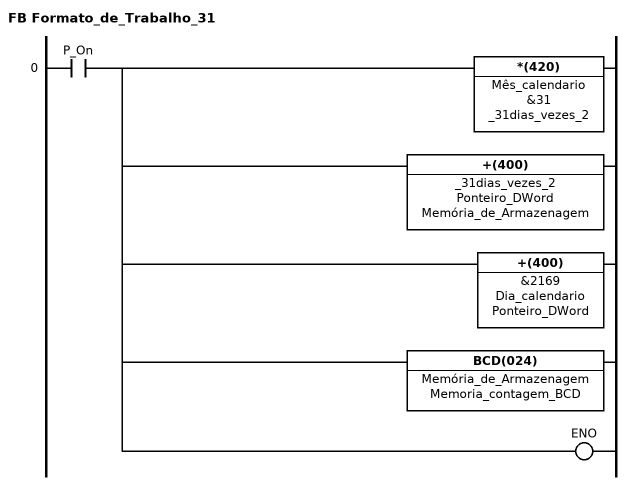
; [picture p48: FB Formato_de_Trabalho_31, rungs 0-0]
; rung 0
LD P_On
*(420) Mês_calendario &31 _31dias_vezes_2
+(400) _31dias_vezes_2 Ponteiro_DWord Memória_de_Armazenagem
+(400) &2169 Dia_calendario Ponteiro_DWord
BCD(024) Memória_de_Armazenagem Memoria_contagem_BCD
OUT ENO